Staubli VAL3: movel_setDO.pgx

public program movel_setDO(point x_pPoint, tool x_tTool, mdesc x_mMdesc, dio& x_dDio)
  local num l_nDist
  local num l_nIndex
  local bool l_bRes
begin

  //execute a movej with the usual arguments (x_pPoint, x_tTool, x_mMdesc) meanwhile
  //when the distance between x_tTool and x_pPoint is lesser than x_nDistance the output x_dDio is set to true

  //the stack is busy
  if bAdvMoves
    l_bRes = watch(!bAdvMoves, nDeadLockTout)
    if !l_bRes
      //it seems stuck!
      call advMovesEmpty(l_bRes)
      //check the "stack" compliance
      call checkAdvMoves()
      if l_bRes
        //but the stack is empty...someone changed it to true manually and saved the library?
        bAdvMoves = false
        libSave()
        logMsg("libSignals/movel_setDO->deadlock fixed")
      endIf
    endIf
  endIf

  setMutex(bAdvMoves)

  if x_mMdesc.blend==off
    l_nDist=nBlendOffToll
  else
    l_nDist=x_mMdesc.leave+nBlendOnToll
  endIf

  //check the "stack" compliance
  call checkAdvMoves()

  //get the first index available
  l_nIndex=-1
  while l_nIndex<0
    call avaAdvMoveIndex(l_nIndex)
    delay(0)
  endWhile

  //get the first index available
  l_nIndex=-1
  while l_nIndex<0
    call avaAdvMoveIndex(l_nIndex)
    delay(0)
  endWhile

  if taskStatus(sAdvMovePrefix+toString("",l_nIndex))==-1
    call lockAdvMove(l_nIndex)
    taskCreate sAdvMovePrefix+toString("",l_nIndex),10,exeMove_setDO(l_nIndex, movel(x_pPoint,x_tTool,x_mMdesc),x_pPoint,x_tTool,l_nDist,x_dDio)
    wait(taskStatus(sAdvMovePrefix+toString("",l_nIndex))==1)
    //launch id watchdog
    call launchIdWD()
  else
    logMsg("libSignals/movel_setDO->error creating the control task")
  endIf

  bAdvMoves = false


end
